(* PLC project Beremiz Python Support Tests, beremiz Beremiz 0.0 *)
(* stored: creationDateTime 2008-12-14T16:21:19, modificationDateTime 2009-09-26T18:14:56 *)

PROGRAM main_pytest
  VAR
    counter : INT;
    DigitalBit0 : BOOL;
    DigitalBit1 : BOOL;
    DigitalBit2 : BOOL;
    DigitalBit3 : BOOL;
    DigitalBit4 : BOOL;
    DigitalBit5 : BOOL;
    DigitalBit6 : BOOL;
    DigitalBit7 : BOOL;
    Start_Stop : Button;
    Compteur : TextCtrl;
    Temoin : Led;
  END_VAR
  VAR  (* added by the conversion: wires and edge detectors of the diagram *)
    _AND96_OUT : BOOL;
    _ADD32_ENO : BOOL;
    _ADD32_OUT : INT;
  END_VAR

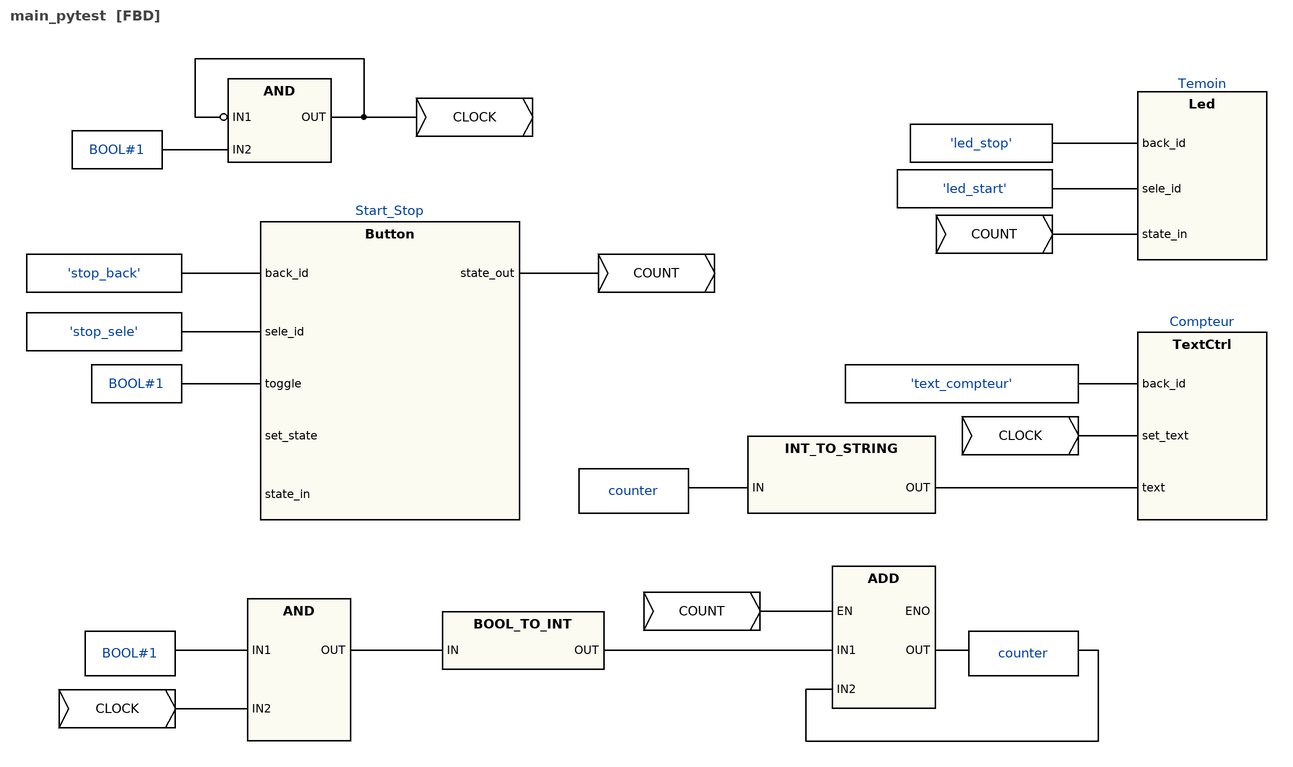
(* FBD diagram, written out as Structured Text *)
Start_Stop(back_id := 'stop_back', sele_id := 'stop_sele', toggle := BOOL#1);
_AND96_OUT := NOT _AND96_OUT AND BOOL#1;
_ADD32_OUT := ADD(EN := Start_Stop.state_out, IN1 := BOOL_TO_INT(BOOL#1 AND _AND96_OUT), IN2 := counter, ENO => _ADD32_ENO);
IF _ADD32_ENO THEN counter := _ADD32_OUT; END_IF;
Temoin(back_id := 'led_stop', sele_id := 'led_start', state_in := Start_Stop.state_out);
Compteur(back_id := 'text_compteur', set_text := _AND96_OUT, text := INT_TO_STRING(counter));
END_PROGRAM

CONFIGURATION conf_pytest
  RESOURCE res_pytest ON PLC
    TASK pytest_task(INTERVAL := t#100ms, PRIORITY := 0);
    PROGRAM pytest_instance : main_pytest;
  END_RESOURCE
END_CONFIGURATION
